FUNCTION_BLOCK Timer0
VAR_INPUT
	bTriggt: BOOL;
END_VAR
VAR
	timer0: ton;
	bQ: BOOL;
END_VAR

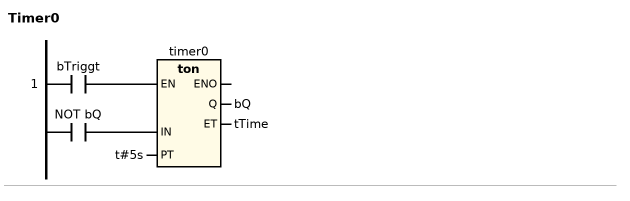
// NETWORK 1
IF bTriggt THEN
    timer0(IN := NOT bQ, PT := t#5s, Q => bQ, ET => tTime); // ton
END_IF

END_FUNCTION_BLOCK

(* stored: Version 1.1.0.1, ProductVersion 3.1.4018.9
   POU Timer0: Id {c439e3c2-519a-4451-baf7-af95d094a96a}, SpecialFunc None *)
